{attribute 'qualified_only'}
{attribute 'strict'}
TYPE E_POP_Type :
(
	EXTEND_CONVEY := 0,
	CONVEY_EXTEND := 1,
	RETRACT_CONVEY := 2,
	CONVEY_RETRACT := 3
);
END_TYPE

(* stored: Version 1.1.0.1, ProductVersion 3.1.4024.12
   DUT E_POP_Type: Id {5a80e3fe-3b38-467a-9c29-53f845bacaba} *)
